// TwinCAT 3 PLC project PLC
// ProgramVersion: 3.1.4024.0
// libraries:
//   SPT Base Types, * (Beckhoff Automation LLC)
//   Tc2_Standard, * (Beckhoff Automation GmbH)
//   Tc2_System, * (Beckhoff Automation GmbH)
//   Tc3_Module, * (Beckhoff Automation GmbH)
//   Tc3_PackML_V2, * (Beckhoff Automation GmbH)
// project tree:
//   DUTs/HMI/ ST_HMI_Machine.TcDUT (not stored), ST_HMI_Machine_Command.TcDUT (not stored), ST_HMI_Machine_Config.TcDUT (not stored), ST_HMI_Machine_Status.TcDUT (not stored)
//   / GlobalTextList.TcGTLO, PlcTask.TcTTO, Visualization Manager.TcVMO (not stored)
//   GVLs/ gHMI.TcGVL
//   POUs/ MAIN.TcPOU
//   Templates/EM/ FB_EM_Template.TcPOU
//   VISUs/VFMs/ VFM_Machine.TcVIS (not stored), VFM_MachineControl.TcVIS (not stored), VFM_Module.TcVIS (not stored), VFM_OperatingMode.TcVIS (not stored), VFM_PackML.TcVIS (not stored), VFM_PackML_Manual.TcVIS (not stored)
//   VISUs/ VIS_Main.TcVIS (not stored)
//   _Machine/00_Machine/ FB_UM_Machine.TcPOU
//   _Machine/01_EM_Infeed/ FB_EM_Infeed.TcPOU
//   _Machine/02_EM_Work/ FB_EM_Work.TcPOU
//   _Machine/03_EM_Outfeed/ FB_EM_Outfeed.TcPOU
// real-time tasks:
//   TASK PlcTask: cycle T#10ms, priority 20, ADS port 350

CONFIGURATION PLC
    RESOURCE PLC ON TwinCAT3
        TASK PlcTask(INTERVAL := T#10ms, PRIORITY := 20);
        PROGRAM MAIN WITH PlcTask : MAIN;
    END_RESOURCE
END_CONFIGURATION

// ---- GVLs/gHMI.TcGVL
{attribute 'qualified_only'}
VAR_GLOBAL
END_VAR

// ---- POUs/MAIN.TcPOU
PROGRAM MAIN
VAR
	Machine: FB_UM_Machine	:= (Name := 'Machine', LogStateChanges := TRUE);
	Initialized: BOOL;
END_VAR

CyclicLogic();

METHOD CyclicLogic : BOOL
VAR_INPUT
END_VAR
IF NOT Initialized THEN
    Initialized := Initialize();
    RETURN;
END_IF

Machine.CyclicLogic();
END_METHOD

METHOD Initialize : BOOL
VAR_INPUT
END_VAR
Initialize := TRUE;
END_METHOD

END_PROGRAM

// ---- _Machine/00_Machine/FB_UM_Machine.TcPOU
FUNCTION_BLOCK FB_UM_Machine EXTENDS FB_PackML_BaseModule
VAR
	// Submodules
	EM_Infeed: 	FB_EM_Infeed 	:= (Name := 'Infeed', LogStateChanges := TRUE);
	EM_Work:	FB_EM_Work 		:= (Name := 'Work', LogStateChanges := TRUE);
	EM_Outfeed:	FB_EM_Outfeed 	:= (Name := 'Outfeed', LogStateChanges := TRUE);
	// Components
	
	// Module Data
	// --Param
	// --Recipe
	// --HMI
	HMI: ST_HMI_Machine;
	
	// Alarms
	
	// Other I/O

	// Machine Control
	rtrigControl: R_TRIG;
	CheckAbort: BOOL;
	CheckStop: BOOL;
	
	// Miscellaneous
	
END_VAR

METHOD PROTECTED Aborted
VAR_INPUT
END_VAR
END_METHOD

METHOD PROTECTED Aborting
VAR_INPUT
END_VAR
CASE _CurrentMode OF
	E_PMLUnitMode.ePMLUnitMode_Production:
        CASE DescendantSequenceState OF
			0:
				NoStateTasksToComplete := FALSE;
				DescendantSequenceState := DescendantSequenceState + 10;
			10:
				StateTasksComplete := TRUE;
		END_CASE
		
	E_PMLUnitMode.ePMLUnitMode_Manual, E_PMLUnitMode.ePMLUnitMode_Maintenance:
        ;	
END_CASE

// Call Super
SUPER^.Aborting();
END_METHOD

METHOD PROTECTED Clearing
VAR_INPUT
END_VAR
CASE _CurrentMode OF
	E_PMLUnitMode.ePMLUnitMode_Production:
        CASE DescendantSequenceState OF
			0:
				NoStateTasksToComplete := FALSE;
				DescendantSequenceState := DescendantSequenceState + 10;
			10:
				StateTasksComplete := TRUE;
		END_CASE
		
	E_PMLUnitMode.ePMLUnitMode_Manual, E_PMLUnitMode.ePMLUnitMode_Maintenance:
        ;	
END_CASE

// Call Super
SUPER^.Clearing();
END_METHOD

METHOD PROTECTED Complete
VAR_INPUT
END_VAR
END_METHOD

//! @summary Initializes event function blocks using this module's name
METHOD PROTECTED CreateEvents

//! @description This method is called by <c>Initialize()</c> as required
// Add your event creation here

// Super call to base
SUPER^.CreateEvents();
END_METHOD

METHOD CyclicLogic
VAR_INPUT
END_VAR
IF NOT _InitComplete THEN
    _InitComplete := Initialize();
    RETURN;
END_IF

MachineControl();

SUPER^.CyclicLogic();
END_METHOD

METHOD PROTECTED Execute
VAR_INPUT
END_VAR
CASE _CurrentMode OF
	E_PMLUnitMode.ePMLUnitMode_Production:
        CASE DescendantSequenceState OF
			0:
				DescendantSequenceState := DescendantSequenceState + 10;
			10:
				;
		END_CASE
		
	E_PMLUnitMode.ePMLUnitMode_Manual, E_PMLUnitMode.ePMLUnitMode_Maintenance:
        ;	
END_CASE
END_METHOD

METHOD PROTECTED Held
VAR_INPUT
END_VAR
END_METHOD

METHOD PROTECTED Holding
VAR_INPUT
END_VAR
CASE _CurrentMode OF
	E_PMLUnitMode.ePMLUnitMode_Production:
        CASE DescendantSequenceState OF
			0:
				NoStateTasksToComplete := FALSE;
				DescendantSequenceState := DescendantSequenceState + 10;
			10:
				StateTasksComplete := TRUE;
		END_CASE
		
	E_PMLUnitMode.ePMLUnitMode_Manual, E_PMLUnitMode.ePMLUnitMode_Maintenance:
        ;	
END_CASE

// Call Super
SUPER^.Holding();
END_METHOD

METHOD PROTECTED Idle
VAR_INPUT
END_VAR
END_METHOD

//! @summary Basic module initialization logic
METHOD PROTECTED Initialize : BOOL;
VAR
	i						 : UDINT;
	varInfo					 : __SYSTEM.VAR_INFO;
	AllSubUnitsInitialized	 : BOOL := TRUE;
	AllComponentsInitialized : BOOL := TRUE;
END_VAR

//! @description This method is called by <c>CyclicLogic()</c> as required
Initialize := FALSE;
CASE DescendantSequenceState OF
    0: // Initialize
        _LogModeChanges         := FALSE;
        _LogStateChanges        := FALSE;
        DescendantSequenceState := DescendantSequenceState + 10;
	
	10: // Register Submodules
		RegisterSubmodule(EM_Infeed);
		RegisterSubmodule(EM_Work);
		RegisterSubmodule(EM_Outfeed);
		DescendantSequenceState := DescendantSequenceState + 10;
		
    20: // Register Components
		//RegisterComponent(component);
        DescendantSequenceState := DescendantSequenceState + 10;
		
    30: // Call the Super
        IF SUPER^.Initialize() THEN
            DescendantSequenceState := DescendantSequenceState + 10;
        END_IF
    40:
        Initialize := TRUE;
END_CASE
END_METHOD

METHOD MachineControl
VAR_INPUT
END_VAR
// Control Triggers
rtrigControl(CLK:= HMI.Command.Start XOR HMI.Command.Stop XOR HMI.Command.Reset XOR HMI.Command.Abort);

CASE CurrentState OF
	E_PMLState.ePMLState_Aborting:
		CheckAbort := FALSE;
		CheckStop := FALSE;
		
	E_PMLState.ePMLState_Aborted:
		// Wait for Reset to Clear
		IF rtrigControl.Q AND HMI.Command.Reset THEN
			ChangeState(E_PMLCommand.ePMLCommand_Clear);
		END_IF
		
	E_PMLState.ePMLState_Clearing:
		CheckAbort := TRUE;
		CheckStop := FALSE;
		
	E_PMLState.ePMLState_Stopping:
		CheckAbort := TRUE;
		CheckStop := FALSE;
		
	E_PMLState.ePMLState_Stopped:
		// Wait for Reset
		IF rtrigControl.Q AND HMI.Command.Reset THEN
			ChangeState(E_PMLCommand.ePMLCommand_Reset);
		END_IF
		
	E_PMLState.ePMLState_Resetting:
		CheckAbort := TRUE;
		CheckStop := TRUE;
	
	E_PMLState.ePMLState_Idle:
		// Wait for Start
		IF rtrigControl.Q AND HMI.Command.Start THEN
			ChangeState(E_PMLCommand.ePMLCommand_Start);
		END_IF
	
END_CASE

// Check for Abort or Stop
IF rtrigControl.Q AND HMI.Command.Abort THEN
	ChangeState(E_PMLCommand.ePMLCommand_Abort);
ELSIF rtrigControl.Q AND HMI.Command.Stop THEN
	ChangeState(E_PMLCommand.ePMLCommand_Stop);
END_IF
END_METHOD

METHOD PROTECTED Resetting
VAR_INPUT
END_VAR
CASE _CurrentMode OF
	E_PMLUnitMode.ePMLUnitMode_Production:
        CASE DescendantSequenceState OF
			0:
				NoStateTasksToComplete := FALSE;
				DescendantSequenceState := DescendantSequenceState + 10;
			10:
				StateTasksComplete := TRUE;
		END_CASE
		
	E_PMLUnitMode.ePMLUnitMode_Manual, E_PMLUnitMode.ePMLUnitMode_Maintenance:
        ;	
END_CASE

// Call Super
SUPER^.Resetting();
END_METHOD

METHOD PROTECTED Starting
VAR_INPUT
END_VAR
CASE _CurrentMode OF
	E_PMLUnitMode.ePMLUnitMode_Production:
        CASE DescendantSequenceState OF
			0:
				NoStateTasksToComplete := FALSE;
				DescendantSequenceState := DescendantSequenceState + 10;
			10:
				StateTasksComplete := TRUE;
		END_CASE
		
	E_PMLUnitMode.ePMLUnitMode_Manual, E_PMLUnitMode.ePMLUnitMode_Maintenance:
        ;	
END_CASE

// Call Super
SUPER^.Starting();
END_METHOD

METHOD PROTECTED Stopped
VAR_INPUT
END_VAR
END_METHOD

METHOD PROTECTED Stopping
VAR_INPUT
END_VAR
CASE _CurrentMode OF
	E_PMLUnitMode.ePMLUnitMode_Production:
        CASE DescendantSequenceState OF
			0:
				NoStateTasksToComplete := FALSE;
				DescendantSequenceState := DescendantSequenceState + 10;
			10:
				StateTasksComplete := TRUE;
		END_CASE
		
	E_PMLUnitMode.ePMLUnitMode_Manual, E_PMLUnitMode.ePMLUnitMode_Maintenance:
        ;	
END_CASE

// Call Super
SUPER^.Stopping();
END_METHOD

METHOD PROTECTED Suspended
VAR_INPUT
END_VAR
END_METHOD

METHOD PROTECTED Suspending
VAR_INPUT
END_VAR
CASE _CurrentMode OF
	E_PMLUnitMode.ePMLUnitMode_Production:
        CASE DescendantSequenceState OF
			0:
				NoStateTasksToComplete := FALSE;
				DescendantSequenceState := DescendantSequenceState + 10;
			10:
				StateTasksComplete := TRUE;
		END_CASE
		
	E_PMLUnitMode.ePMLUnitMode_Manual, E_PMLUnitMode.ePMLUnitMode_Maintenance:
        ;	
END_CASE

// Call Super
SUPER^.Suspending();
END_METHOD

METHOD PROTECTED Undefined
VAR_INPUT
END_VAR
END_METHOD

METHOD PROTECTED Unholding
VAR_INPUT
END_VAR
CASE _CurrentMode OF
	E_PMLUnitMode.ePMLUnitMode_Production:
        CASE DescendantSequenceState OF
			0:
				NoStateTasksToComplete := FALSE;
				DescendantSequenceState := DescendantSequenceState + 10;
			10:
				StateTasksComplete := TRUE;
		END_CASE
		
	E_PMLUnitMode.ePMLUnitMode_Manual, E_PMLUnitMode.ePMLUnitMode_Maintenance:
        ;	
END_CASE

// Call Super
SUPER^.Unholding();
END_METHOD

METHOD PROTECTED Unsuspending
VAR_INPUT
END_VAR
CASE _CurrentMode OF
	E_PMLUnitMode.ePMLUnitMode_Production:
        CASE DescendantSequenceState OF
			0:
				NoStateTasksToComplete := FALSE;
				DescendantSequenceState := DescendantSequenceState + 10;
			10:
				StateTasksComplete := TRUE;
		END_CASE
		
	E_PMLUnitMode.ePMLUnitMode_Manual, E_PMLUnitMode.ePMLUnitMode_Maintenance:
        ;	
END_CASE

// Call Super
SUPER^.Unsuspending();
END_METHOD

END_FUNCTION_BLOCK

// ---- _Machine/01_EM_Infeed/FB_EM_Infeed.TcPOU
FUNCTION_BLOCK FB_EM_Infeed EXTENDS FB_PackML_BaseModule
VAR
	// Submodules
	
	// Components
	
	// Module Data
	// --Param
	// --Recipe
	// --HMI
	
	// Alarms
	
	// Other I/O
	
	// Miscellaneous
	
END_VAR

METHOD PROTECTED Aborted
VAR_INPUT
END_VAR
END_METHOD

METHOD PROTECTED Aborting
VAR_INPUT
END_VAR
CASE _CurrentMode OF
	E_PMLUnitMode.ePMLUnitMode_Production:
        CASE DescendantSequenceState OF
			0:
				NoStateTasksToComplete := FALSE;
				DescendantSequenceState := DescendantSequenceState + 10;
			10:
				StateTasksComplete := TRUE;
		END_CASE
		
	E_PMLUnitMode.ePMLUnitMode_Manual, E_PMLUnitMode.ePMLUnitMode_Maintenance:
        ;	
END_CASE

// Call Super
SUPER^.Aborting();
END_METHOD

METHOD PROTECTED Clearing
VAR_INPUT
END_VAR
CASE _CurrentMode OF
	E_PMLUnitMode.ePMLUnitMode_Production:
        CASE DescendantSequenceState OF
			0:
				NoStateTasksToComplete := FALSE;
				DescendantSequenceState := DescendantSequenceState + 10;
			10:
				StateTasksComplete := TRUE;
		END_CASE
		
	E_PMLUnitMode.ePMLUnitMode_Manual, E_PMLUnitMode.ePMLUnitMode_Maintenance:
        ;	
END_CASE

// Call Super
SUPER^.Clearing();
END_METHOD

METHOD PROTECTED Complete
VAR_INPUT
END_VAR
END_METHOD

//! @summary Initializes event function blocks using this module's name
METHOD PROTECTED CreateEvents

//! @description This method is called by <c>Initialize()</c> as required
// Add your event creation here

// Super call to base
SUPER^.CreateEvents();
END_METHOD

METHOD CyclicLogic
VAR_INPUT
END_VAR
IF NOT _InitComplete THEN
    _InitComplete := Initialize();
    RETURN;
END_IF

SUPER^.CyclicLogic();
END_METHOD

METHOD PROTECTED Execute
VAR_INPUT
END_VAR
CASE _CurrentMode OF
	E_PMLUnitMode.ePMLUnitMode_Production:
        CASE DescendantSequenceState OF
			0:
				DescendantSequenceState := DescendantSequenceState + 10;
			10:
				;
		END_CASE
		
	E_PMLUnitMode.ePMLUnitMode_Manual, E_PMLUnitMode.ePMLUnitMode_Maintenance:
        ;	
END_CASE
END_METHOD

METHOD PROTECTED Held
VAR_INPUT
END_VAR
END_METHOD

METHOD PROTECTED Holding
VAR_INPUT
END_VAR
CASE _CurrentMode OF
	E_PMLUnitMode.ePMLUnitMode_Production:
        CASE DescendantSequenceState OF
			0:
				NoStateTasksToComplete := FALSE;
				DescendantSequenceState := DescendantSequenceState + 10;
			10:
				StateTasksComplete := TRUE;
		END_CASE
		
	E_PMLUnitMode.ePMLUnitMode_Manual, E_PMLUnitMode.ePMLUnitMode_Maintenance:
        ;	
END_CASE

// Call Super
SUPER^.Holding();
END_METHOD

METHOD PROTECTED Idle
VAR_INPUT
END_VAR
END_METHOD

//! @summary Basic module initialization logic
METHOD PROTECTED Initialize : BOOL;
VAR
	i						 : UDINT;
	varInfo					 : __SYSTEM.VAR_INFO;
	AllSubUnitsInitialized	 : BOOL := TRUE;
	AllComponentsInitialized : BOOL := TRUE;
END_VAR

//! @description This method is called by <c>CyclicLogic()</c> as required
Initialize := FALSE;
CASE DescendantSequenceState OF
    0: // Initialize
        _LogModeChanges         := FALSE;
        _LogStateChanges        := FALSE;
        DescendantSequenceState := DescendantSequenceState + 10;
	
	10: // Register Submodules
		//RegisterSubmodule(submodule);
		DescendantSequenceState := DescendantSequenceState + 10;
    20: // Register Components
		//RegisterComponent(component);
        DescendantSequenceState := DescendantSequenceState + 10;
    30: // Call the Super
        IF SUPER^.Initialize() THEN
            DescendantSequenceState := DescendantSequenceState + 10;
        END_IF
    40:
        Initialize := TRUE;
END_CASE
END_METHOD

METHOD PROTECTED Resetting
VAR_INPUT
END_VAR
CASE _CurrentMode OF
	E_PMLUnitMode.ePMLUnitMode_Production:
        CASE DescendantSequenceState OF
			0:
				NoStateTasksToComplete := FALSE;
				DescendantSequenceState := DescendantSequenceState + 10;
			10:
				StateTasksComplete := TRUE;
		END_CASE
		
	E_PMLUnitMode.ePMLUnitMode_Manual, E_PMLUnitMode.ePMLUnitMode_Maintenance:
        ;	
END_CASE

// Call Super
SUPER^.Resetting();
END_METHOD

METHOD PROTECTED Starting
VAR_INPUT
END_VAR
CASE _CurrentMode OF
	E_PMLUnitMode.ePMLUnitMode_Production:
        CASE DescendantSequenceState OF
			0:
				NoStateTasksToComplete := FALSE;
				DescendantSequenceState := DescendantSequenceState + 10;
			10:
				StateTasksComplete := TRUE;
		END_CASE
		
	E_PMLUnitMode.ePMLUnitMode_Manual, E_PMLUnitMode.ePMLUnitMode_Maintenance:
        ;	
END_CASE

// Call Super
SUPER^.Starting();
END_METHOD

METHOD PROTECTED Stopped
VAR_INPUT
END_VAR
END_METHOD

METHOD PROTECTED Stopping
VAR_INPUT
END_VAR
CASE _CurrentMode OF
	E_PMLUnitMode.ePMLUnitMode_Production:
        CASE DescendantSequenceState OF
			0:
				NoStateTasksToComplete := FALSE;
				DescendantSequenceState := DescendantSequenceState + 10;
			10:
				StateTasksComplete := TRUE;
		END_CASE
		
	E_PMLUnitMode.ePMLUnitMode_Manual, E_PMLUnitMode.ePMLUnitMode_Maintenance:
        ;	
END_CASE

// Call Super
SUPER^.Stopping();
END_METHOD

METHOD PROTECTED Suspended
VAR_INPUT
END_VAR
END_METHOD

METHOD PROTECTED Suspending
VAR_INPUT
END_VAR
CASE _CurrentMode OF
	E_PMLUnitMode.ePMLUnitMode_Production:
        CASE DescendantSequenceState OF
			0:
				NoStateTasksToComplete := FALSE;
				DescendantSequenceState := DescendantSequenceState + 10;
			10:
				StateTasksComplete := TRUE;
		END_CASE
		
	E_PMLUnitMode.ePMLUnitMode_Manual, E_PMLUnitMode.ePMLUnitMode_Maintenance:
        ;	
END_CASE

// Call Super
SUPER^.Suspending();
END_METHOD

METHOD PROTECTED Undefined
VAR_INPUT
END_VAR
END_METHOD

METHOD PROTECTED Unholding
VAR_INPUT
END_VAR
CASE _CurrentMode OF
	E_PMLUnitMode.ePMLUnitMode_Production:
        CASE DescendantSequenceState OF
			0:
				NoStateTasksToComplete := FALSE;
				DescendantSequenceState := DescendantSequenceState + 10;
			10:
				StateTasksComplete := TRUE;
		END_CASE
		
	E_PMLUnitMode.ePMLUnitMode_Manual, E_PMLUnitMode.ePMLUnitMode_Maintenance:
        ;	
END_CASE

// Call Super
SUPER^.Unholding();
END_METHOD

METHOD PROTECTED Unsuspending
VAR_INPUT
END_VAR
CASE _CurrentMode OF
	E_PMLUnitMode.ePMLUnitMode_Production:
        CASE DescendantSequenceState OF
			0:
				NoStateTasksToComplete := FALSE;
				DescendantSequenceState := DescendantSequenceState + 10;
			10:
				StateTasksComplete := TRUE;
		END_CASE
		
	E_PMLUnitMode.ePMLUnitMode_Manual, E_PMLUnitMode.ePMLUnitMode_Maintenance:
        ;	
END_CASE

// Call Super
SUPER^.Unsuspending();
END_METHOD

END_FUNCTION_BLOCK

// ---- _Machine/02_EM_Work/FB_EM_Work.TcPOU
FUNCTION_BLOCK FB_EM_Work EXTENDS FB_PackML_BaseModule
VAR
	// Submodules
	
	// Components
	
	// Module Data
	// --Param
	// --Recipe
	// --HMI
	
	// Alarms
	
	// Other I/O
	
	// Miscellaneous
	
END_VAR

METHOD PROTECTED Aborted
VAR_INPUT
END_VAR
END_METHOD

METHOD PROTECTED Aborting
VAR_INPUT
END_VAR
CASE _CurrentMode OF
	E_PMLUnitMode.ePMLUnitMode_Production:
        CASE DescendantSequenceState OF
			0:
				NoStateTasksToComplete := FALSE;
				DescendantSequenceState := DescendantSequenceState + 10;
			10:
				StateTasksComplete := TRUE;
		END_CASE
		
	E_PMLUnitMode.ePMLUnitMode_Manual, E_PMLUnitMode.ePMLUnitMode_Maintenance:
        ;	
END_CASE

// Call Super
SUPER^.Aborting();
END_METHOD

METHOD PROTECTED Clearing
VAR_INPUT
END_VAR
CASE _CurrentMode OF
	E_PMLUnitMode.ePMLUnitMode_Production:
        CASE DescendantSequenceState OF
			0:
				NoStateTasksToComplete := FALSE;
				DescendantSequenceState := DescendantSequenceState + 10;
			10:
				StateTasksComplete := TRUE;
		END_CASE
		
	E_PMLUnitMode.ePMLUnitMode_Manual, E_PMLUnitMode.ePMLUnitMode_Maintenance:
        ;	
END_CASE

// Call Super
SUPER^.Clearing();
END_METHOD

METHOD PROTECTED Complete
VAR_INPUT
END_VAR
END_METHOD

//! @summary Initializes event function blocks using this module's name
METHOD PROTECTED CreateEvents

//! @description This method is called by <c>Initialize()</c> as required
// Add your event creation here

// Super call to base
SUPER^.CreateEvents();
END_METHOD

METHOD CyclicLogic
VAR_INPUT
END_VAR
IF NOT _InitComplete THEN
    _InitComplete := Initialize();
    RETURN;
END_IF

SUPER^.CyclicLogic();
END_METHOD

METHOD PROTECTED Execute
VAR_INPUT
END_VAR
CASE _CurrentMode OF
	E_PMLUnitMode.ePMLUnitMode_Production:
        CASE DescendantSequenceState OF
			0:
				DescendantSequenceState := DescendantSequenceState + 10;
			10:
				;
		END_CASE
		
	E_PMLUnitMode.ePMLUnitMode_Manual, E_PMLUnitMode.ePMLUnitMode_Maintenance:
        ;	
END_CASE
END_METHOD

METHOD PROTECTED Held
VAR_INPUT
END_VAR
END_METHOD

METHOD PROTECTED Holding
VAR_INPUT
END_VAR
CASE _CurrentMode OF
	E_PMLUnitMode.ePMLUnitMode_Production:
        CASE DescendantSequenceState OF
			0:
				NoStateTasksToComplete := FALSE;
				DescendantSequenceState := DescendantSequenceState + 10;
			10:
				StateTasksComplete := TRUE;
		END_CASE
		
	E_PMLUnitMode.ePMLUnitMode_Manual, E_PMLUnitMode.ePMLUnitMode_Maintenance:
        ;	
END_CASE

// Call Super
SUPER^.Holding();
END_METHOD

METHOD PROTECTED Idle
VAR_INPUT
END_VAR
END_METHOD

//! @summary Basic module initialization logic
METHOD PROTECTED Initialize : BOOL;
VAR
	i						 : UDINT;
	varInfo					 : __SYSTEM.VAR_INFO;
	AllSubUnitsInitialized	 : BOOL := TRUE;
	AllComponentsInitialized : BOOL := TRUE;
END_VAR

//! @description This method is called by <c>CyclicLogic()</c> as required
Initialize := FALSE;
CASE DescendantSequenceState OF
    0: // Initialize
        _LogModeChanges         := FALSE;
        _LogStateChanges        := FALSE;
        DescendantSequenceState := DescendantSequenceState + 10;
	
	10: // Register Submodules
		//RegisterSubmodule(submodule);
		DescendantSequenceState := DescendantSequenceState + 10;
    20: // Register Components
		//RegisterComponent(component);
        DescendantSequenceState := DescendantSequenceState + 10;
    30: // Call the Super
        IF SUPER^.Initialize() THEN
            DescendantSequenceState := DescendantSequenceState + 10;
        END_IF
    40:
        Initialize := TRUE;
END_CASE
END_METHOD

METHOD PROTECTED Resetting
VAR_INPUT
END_VAR
CASE _CurrentMode OF
	E_PMLUnitMode.ePMLUnitMode_Production:
        CASE DescendantSequenceState OF
			0:
				NoStateTasksToComplete := FALSE;
				DescendantSequenceState := DescendantSequenceState + 10;
			10:
				StateTasksComplete := TRUE;
		END_CASE
		
	E_PMLUnitMode.ePMLUnitMode_Manual, E_PMLUnitMode.ePMLUnitMode_Maintenance:
        ;	
END_CASE

// Call Super
SUPER^.Resetting();
END_METHOD

METHOD PROTECTED Starting
VAR_INPUT
END_VAR
CASE _CurrentMode OF
	E_PMLUnitMode.ePMLUnitMode_Production:
        CASE DescendantSequenceState OF
			0:
				NoStateTasksToComplete := FALSE;
				DescendantSequenceState := DescendantSequenceState + 10;
			10:
				StateTasksComplete := TRUE;
		END_CASE
		
	E_PMLUnitMode.ePMLUnitMode_Manual, E_PMLUnitMode.ePMLUnitMode_Maintenance:
        ;	
END_CASE

// Call Super
SUPER^.Starting();
END_METHOD

METHOD PROTECTED Stopped
VAR_INPUT
END_VAR
END_METHOD

METHOD PROTECTED Stopping
VAR_INPUT
END_VAR
CASE _CurrentMode OF
	E_PMLUnitMode.ePMLUnitMode_Production:
        CASE DescendantSequenceState OF
			0:
				NoStateTasksToComplete := FALSE;
				DescendantSequenceState := DescendantSequenceState + 10;
			10:
				StateTasksComplete := TRUE;
		END_CASE
		
	E_PMLUnitMode.ePMLUnitMode_Manual, E_PMLUnitMode.ePMLUnitMode_Maintenance:
        ;	
END_CASE

// Call Super
SUPER^.Stopping();
END_METHOD

METHOD PROTECTED Suspended
VAR_INPUT
END_VAR
END_METHOD

METHOD PROTECTED Suspending
VAR_INPUT
END_VAR
CASE _CurrentMode OF
	E_PMLUnitMode.ePMLUnitMode_Production:
        CASE DescendantSequenceState OF
			0:
				NoStateTasksToComplete := FALSE;
				DescendantSequenceState := DescendantSequenceState + 10;
			10:
				StateTasksComplete := TRUE;
		END_CASE
		
	E_PMLUnitMode.ePMLUnitMode_Manual, E_PMLUnitMode.ePMLUnitMode_Maintenance:
        ;	
END_CASE

// Call Super
SUPER^.Suspending();
END_METHOD

METHOD PROTECTED Undefined
VAR_INPUT
END_VAR
END_METHOD

METHOD PROTECTED Unholding
VAR_INPUT
END_VAR
CASE _CurrentMode OF
	E_PMLUnitMode.ePMLUnitMode_Production:
        CASE DescendantSequenceState OF
			0:
				NoStateTasksToComplete := FALSE;
				DescendantSequenceState := DescendantSequenceState + 10;
			10:
				StateTasksComplete := TRUE;
		END_CASE
		
	E_PMLUnitMode.ePMLUnitMode_Manual, E_PMLUnitMode.ePMLUnitMode_Maintenance:
        ;	
END_CASE

// Call Super
SUPER^.Unholding();
END_METHOD

METHOD PROTECTED Unsuspending
VAR_INPUT
END_VAR
CASE _CurrentMode OF
	E_PMLUnitMode.ePMLUnitMode_Production:
        CASE DescendantSequenceState OF
			0:
				NoStateTasksToComplete := FALSE;
				DescendantSequenceState := DescendantSequenceState + 10;
			10:
				StateTasksComplete := TRUE;
		END_CASE
		
	E_PMLUnitMode.ePMLUnitMode_Manual, E_PMLUnitMode.ePMLUnitMode_Maintenance:
        ;	
END_CASE

// Call Super
SUPER^.Unsuspending();
END_METHOD

END_FUNCTION_BLOCK

// ---- _Machine/03_EM_Outfeed/FB_EM_Outfeed.TcPOU
FUNCTION_BLOCK FB_EM_Outfeed EXTENDS FB_PackML_BaseModule
VAR
	// Submodules
	
	// Components
	
	// Module Data
	// --Param
	// --Recipe
	// --HMI
	
	// Alarms
	
	// Other I/O
	
	// Miscellaneous
	
END_VAR

METHOD PROTECTED Aborted
VAR_INPUT
END_VAR
END_METHOD

METHOD PROTECTED Aborting
VAR_INPUT
END_VAR
CASE _CurrentMode OF
	E_PMLUnitMode.ePMLUnitMode_Production:
        CASE DescendantSequenceState OF
			0:
				NoStateTasksToComplete := FALSE;
				DescendantSequenceState := DescendantSequenceState + 10;
			10:
				StateTasksComplete := TRUE;
		END_CASE
		
	E_PMLUnitMode.ePMLUnitMode_Manual, E_PMLUnitMode.ePMLUnitMode_Maintenance:
        ;	
END_CASE

// Call Super
SUPER^.Aborting();
END_METHOD

METHOD PROTECTED Clearing
VAR_INPUT
END_VAR
CASE _CurrentMode OF
	E_PMLUnitMode.ePMLUnitMode_Production:
        CASE DescendantSequenceState OF
			0:
				NoStateTasksToComplete := FALSE;
				DescendantSequenceState := DescendantSequenceState + 10;
			10:
				StateTasksComplete := TRUE;
		END_CASE
		
	E_PMLUnitMode.ePMLUnitMode_Manual, E_PMLUnitMode.ePMLUnitMode_Maintenance:
        ;	
END_CASE

// Call Super
SUPER^.Clearing();
END_METHOD

METHOD PROTECTED Complete
VAR_INPUT
END_VAR
END_METHOD

//! @summary Initializes event function blocks using this module's name
METHOD PROTECTED CreateEvents

//! @description This method is called by <c>Initialize()</c> as required
// Add your event creation here

// Super call to base
SUPER^.CreateEvents();
END_METHOD

METHOD CyclicLogic
VAR_INPUT
END_VAR
IF NOT _InitComplete THEN
    _InitComplete := Initialize();
    RETURN;
END_IF

SUPER^.CyclicLogic();
END_METHOD

METHOD PROTECTED Execute
VAR_INPUT
END_VAR
CASE _CurrentMode OF
	E_PMLUnitMode.ePMLUnitMode_Production:
        CASE DescendantSequenceState OF
			0:
				DescendantSequenceState := DescendantSequenceState + 10;
			10:
				;
		END_CASE
		
	E_PMLUnitMode.ePMLUnitMode_Manual, E_PMLUnitMode.ePMLUnitMode_Maintenance:
        ;	
END_CASE
END_METHOD

METHOD PROTECTED Held
VAR_INPUT
END_VAR
END_METHOD

METHOD PROTECTED Holding
VAR_INPUT
END_VAR
CASE _CurrentMode OF
	E_PMLUnitMode.ePMLUnitMode_Production:
        CASE DescendantSequenceState OF
			0:
				NoStateTasksToComplete := FALSE;
				DescendantSequenceState := DescendantSequenceState + 10;
			10:
				StateTasksComplete := TRUE;
		END_CASE
		
	E_PMLUnitMode.ePMLUnitMode_Manual, E_PMLUnitMode.ePMLUnitMode_Maintenance:
        ;	
END_CASE

// Call Super
SUPER^.Holding();
END_METHOD

METHOD PROTECTED Idle
VAR_INPUT
END_VAR
END_METHOD

//! @summary Basic module initialization logic
METHOD PROTECTED Initialize : BOOL;
VAR
	i						 : UDINT;
	varInfo					 : __SYSTEM.VAR_INFO;
	AllSubUnitsInitialized	 : BOOL := TRUE;
	AllComponentsInitialized : BOOL := TRUE;
END_VAR

//! @description This method is called by <c>CyclicLogic()</c> as required
Initialize := FALSE;
CASE DescendantSequenceState OF
    0: // Initialize
        _LogModeChanges         := FALSE;
        _LogStateChanges        := FALSE;
        DescendantSequenceState := DescendantSequenceState + 10;
	
	10: // Register Submodules
		//RegisterSubmodule(submodule);
		DescendantSequenceState := DescendantSequenceState + 10;
    20: // Register Components
		//RegisterComponent(component);
        DescendantSequenceState := DescendantSequenceState + 10;
    30: // Call the Super
        IF SUPER^.Initialize() THEN
            DescendantSequenceState := DescendantSequenceState + 10;
        END_IF
    40:
        Initialize := TRUE;
END_CASE
END_METHOD

METHOD PROTECTED Resetting
VAR_INPUT
END_VAR
CASE _CurrentMode OF
	E_PMLUnitMode.ePMLUnitMode_Production:
        CASE DescendantSequenceState OF
			0:
				NoStateTasksToComplete := FALSE;
				DescendantSequenceState := DescendantSequenceState + 10;
			10:
				StateTasksComplete := TRUE;
		END_CASE
		
	E_PMLUnitMode.ePMLUnitMode_Manual, E_PMLUnitMode.ePMLUnitMode_Maintenance:
        ;	
END_CASE

// Call Super
SUPER^.Resetting();
END_METHOD

METHOD PROTECTED Starting
VAR_INPUT
END_VAR
CASE _CurrentMode OF
	E_PMLUnitMode.ePMLUnitMode_Production:
        CASE DescendantSequenceState OF
			0:
				NoStateTasksToComplete := FALSE;
				DescendantSequenceState := DescendantSequenceState + 10;
			10:
				StateTasksComplete := TRUE;
		END_CASE
		
	E_PMLUnitMode.ePMLUnitMode_Manual, E_PMLUnitMode.ePMLUnitMode_Maintenance:
        ;	
END_CASE

// Call Super
SUPER^.Starting();
END_METHOD

METHOD PROTECTED Stopped
VAR_INPUT
END_VAR
END_METHOD

METHOD PROTECTED Stopping
VAR_INPUT
END_VAR
CASE _CurrentMode OF
	E_PMLUnitMode.ePMLUnitMode_Production:
        CASE DescendantSequenceState OF
			0:
				NoStateTasksToComplete := FALSE;
				DescendantSequenceState := DescendantSequenceState + 10;
			10:
				StateTasksComplete := TRUE;
		END_CASE
		
	E_PMLUnitMode.ePMLUnitMode_Manual, E_PMLUnitMode.ePMLUnitMode_Maintenance:
        ;	
END_CASE

// Call Super
SUPER^.Stopping();
END_METHOD

METHOD PROTECTED Suspended
VAR_INPUT
END_VAR
END_METHOD

METHOD PROTECTED Suspending
VAR_INPUT
END_VAR
CASE _CurrentMode OF
	E_PMLUnitMode.ePMLUnitMode_Production:
        CASE DescendantSequenceState OF
			0:
				NoStateTasksToComplete := FALSE;
				DescendantSequenceState := DescendantSequenceState + 10;
			10:
				StateTasksComplete := TRUE;
		END_CASE
		
	E_PMLUnitMode.ePMLUnitMode_Manual, E_PMLUnitMode.ePMLUnitMode_Maintenance:
        ;	
END_CASE

// Call Super
SUPER^.Suspending();
END_METHOD

METHOD PROTECTED Undefined
VAR_INPUT
END_VAR
END_METHOD

METHOD PROTECTED Unholding
VAR_INPUT
END_VAR
CASE _CurrentMode OF
	E_PMLUnitMode.ePMLUnitMode_Production:
        CASE DescendantSequenceState OF
			0:
				NoStateTasksToComplete := FALSE;
				DescendantSequenceState := DescendantSequenceState + 10;
			10:
				StateTasksComplete := TRUE;
		END_CASE
		
	E_PMLUnitMode.ePMLUnitMode_Manual, E_PMLUnitMode.ePMLUnitMode_Maintenance:
        ;	
END_CASE

// Call Super
SUPER^.Unholding();
END_METHOD

METHOD PROTECTED Unsuspending
VAR_INPUT
END_VAR
CASE _CurrentMode OF
	E_PMLUnitMode.ePMLUnitMode_Production:
        CASE DescendantSequenceState OF
			0:
				NoStateTasksToComplete := FALSE;
				DescendantSequenceState := DescendantSequenceState + 10;
			10:
				StateTasksComplete := TRUE;
		END_CASE
		
	E_PMLUnitMode.ePMLUnitMode_Manual, E_PMLUnitMode.ePMLUnitMode_Maintenance:
        ;	
END_CASE

// Call Super
SUPER^.Unsuspending();
END_METHOD

END_FUNCTION_BLOCK

// ---- Templates/EM/FB_EM_Template.TcPOU
FUNCTION_BLOCK FB_EM_Template EXTENDS FB_PackML_BaseModule
VAR
	// Submodules
	
	// Components
	
	// Module Data
	// --Param
	// --Recipe
	// --HMI
	
	// Alarms
	
	// Other I/O
	
	// Miscellaneous
	
END_VAR

METHOD PROTECTED Aborted
VAR_INPUT
END_VAR
END_METHOD

METHOD PROTECTED Aborting
VAR_INPUT
END_VAR
CASE _CurrentMode OF
	E_PMLUnitMode.ePMLUnitMode_Production:
        CASE DescendantSequenceState OF
			0:
				NoStateTasksToComplete := FALSE;
				DescendantSequenceState := DescendantSequenceState + 10;
			10:
				StateTasksComplete := TRUE;
		END_CASE
		
	E_PMLUnitMode.ePMLUnitMode_Manual, E_PMLUnitMode.ePMLUnitMode_Maintenance:
        ;	
END_CASE

// Call Super
SUPER^.Aborting();
END_METHOD

METHOD PROTECTED Clearing
VAR_INPUT
END_VAR
CASE _CurrentMode OF
	E_PMLUnitMode.ePMLUnitMode_Production:
        CASE DescendantSequenceState OF
			0:
				NoStateTasksToComplete := FALSE;
				DescendantSequenceState := DescendantSequenceState + 10;
			10:
				StateTasksComplete := TRUE;
		END_CASE
		
	E_PMLUnitMode.ePMLUnitMode_Manual, E_PMLUnitMode.ePMLUnitMode_Maintenance:
        ;	
END_CASE

// Call Super
SUPER^.Clearing();
END_METHOD

METHOD PROTECTED Complete
VAR_INPUT
END_VAR
END_METHOD

//! @summary Initializes event function blocks using this module's name
METHOD PROTECTED CreateEvents

//! @description This method is called by <c>Initialize()</c> as required
// Add your event creation here

// Super call to base
SUPER^.CreateEvents();
END_METHOD

METHOD CyclicLogic
VAR_INPUT
END_VAR
IF NOT _InitComplete THEN
    _InitComplete := Initialize();
    RETURN;
END_IF

SUPER^.CyclicLogic();
END_METHOD

METHOD PROTECTED Execute
VAR_INPUT
END_VAR
CASE _CurrentMode OF
	E_PMLUnitMode.ePMLUnitMode_Production:
        CASE DescendantSequenceState OF
			0:
				DescendantSequenceState := DescendantSequenceState + 10;
			10:
				;
		END_CASE
		
	E_PMLUnitMode.ePMLUnitMode_Manual, E_PMLUnitMode.ePMLUnitMode_Maintenance:
        ;	
END_CASE
END_METHOD

METHOD PROTECTED Held
VAR_INPUT
END_VAR
END_METHOD

METHOD PROTECTED Holding
VAR_INPUT
END_VAR
CASE _CurrentMode OF
	E_PMLUnitMode.ePMLUnitMode_Production:
        CASE DescendantSequenceState OF
			0:
				NoStateTasksToComplete := FALSE;
				DescendantSequenceState := DescendantSequenceState + 10;
			10:
				StateTasksComplete := TRUE;
		END_CASE
		
	E_PMLUnitMode.ePMLUnitMode_Manual, E_PMLUnitMode.ePMLUnitMode_Maintenance:
        ;	
END_CASE

// Call Super
SUPER^.Holding();
END_METHOD

METHOD PROTECTED Idle
VAR_INPUT
END_VAR
END_METHOD

//! @summary Basic module initialization logic
METHOD PROTECTED Initialize : BOOL;
VAR
	i						 : UDINT;
	varInfo					 : __SYSTEM.VAR_INFO;
	AllSubUnitsInitialized	 : BOOL := TRUE;
	AllComponentsInitialized : BOOL := TRUE;
END_VAR

//! @description This method is called by <c>CyclicLogic()</c> as required
Initialize := FALSE;
CASE DescendantSequenceState OF
    0: // Initialize
        _LogModeChanges         := FALSE;
        _LogStateChanges        := FALSE;
        DescendantSequenceState := DescendantSequenceState + 10;
	
	10: // Register Submodules
		//RegisterSubmodule(submodule);
		DescendantSequenceState := DescendantSequenceState + 10;
    20: // Register Components
		//RegisterComponent(component);
        DescendantSequenceState := DescendantSequenceState + 10;
    30: // Call the Super
        IF SUPER^.Initialize() THEN
            DescendantSequenceState := DescendantSequenceState + 10;
        END_IF
    40:
        Initialize := TRUE;
END_CASE
END_METHOD

METHOD PROTECTED Resetting
VAR_INPUT
END_VAR
CASE _CurrentMode OF
	E_PMLUnitMode.ePMLUnitMode_Production:
        CASE DescendantSequenceState OF
			0:
				NoStateTasksToComplete := FALSE;
				DescendantSequenceState := DescendantSequenceState + 10;
			10:
				StateTasksComplete := TRUE;
		END_CASE
		
	E_PMLUnitMode.ePMLUnitMode_Manual, E_PMLUnitMode.ePMLUnitMode_Maintenance:
        ;	
END_CASE

// Call Super
SUPER^.Resetting();
END_METHOD

METHOD PROTECTED Starting
VAR_INPUT
END_VAR
CASE _CurrentMode OF
	E_PMLUnitMode.ePMLUnitMode_Production:
        CASE DescendantSequenceState OF
			0:
				NoStateTasksToComplete := FALSE;
				DescendantSequenceState := DescendantSequenceState + 10;
			10:
				StateTasksComplete := TRUE;
		END_CASE
		
	E_PMLUnitMode.ePMLUnitMode_Manual, E_PMLUnitMode.ePMLUnitMode_Maintenance:
        ;	
END_CASE

// Call Super
SUPER^.Starting();
END_METHOD

METHOD PROTECTED Stopped
VAR_INPUT
END_VAR
END_METHOD

METHOD PROTECTED Stopping
VAR_INPUT
END_VAR
CASE _CurrentMode OF
	E_PMLUnitMode.ePMLUnitMode_Production:
        CASE DescendantSequenceState OF
			0:
				NoStateTasksToComplete := FALSE;
				DescendantSequenceState := DescendantSequenceState + 10;
			10:
				StateTasksComplete := TRUE;
		END_CASE
		
	E_PMLUnitMode.ePMLUnitMode_Manual, E_PMLUnitMode.ePMLUnitMode_Maintenance:
        ;	
END_CASE

// Call Super
SUPER^.Stopping();
END_METHOD

METHOD PROTECTED Suspended
VAR_INPUT
END_VAR
END_METHOD

METHOD PROTECTED Suspending
VAR_INPUT
END_VAR
CASE _CurrentMode OF
	E_PMLUnitMode.ePMLUnitMode_Production:
        CASE DescendantSequenceState OF
			0:
				NoStateTasksToComplete := FALSE;
				DescendantSequenceState := DescendantSequenceState + 10;
			10:
				StateTasksComplete := TRUE;
		END_CASE
		
	E_PMLUnitMode.ePMLUnitMode_Manual, E_PMLUnitMode.ePMLUnitMode_Maintenance:
        ;	
END_CASE

// Call Super
SUPER^.Suspending();
END_METHOD

METHOD PROTECTED Undefined
VAR_INPUT
END_VAR
END_METHOD

METHOD PROTECTED Unholding
VAR_INPUT
END_VAR
CASE _CurrentMode OF
	E_PMLUnitMode.ePMLUnitMode_Production:
        CASE DescendantSequenceState OF
			0:
				NoStateTasksToComplete := FALSE;
				DescendantSequenceState := DescendantSequenceState + 10;
			10:
				StateTasksComplete := TRUE;
		END_CASE
		
	E_PMLUnitMode.ePMLUnitMode_Manual, E_PMLUnitMode.ePMLUnitMode_Maintenance:
        ;	
END_CASE

// Call Super
SUPER^.Unholding();
END_METHOD

METHOD PROTECTED Unsuspending
VAR_INPUT
END_VAR
CASE _CurrentMode OF
	E_PMLUnitMode.ePMLUnitMode_Production:
        CASE DescendantSequenceState OF
			0:
				NoStateTasksToComplete := FALSE;
				DescendantSequenceState := DescendantSequenceState + 10;
			10:
				StateTasksComplete := TRUE;
		END_CASE
		
	E_PMLUnitMode.ePMLUnitMode_Manual, E_PMLUnitMode.ePMLUnitMode_Maintenance:
        ;	
END_CASE

// Call Super
SUPER^.Unsuspending();
END_METHOD

END_FUNCTION_BLOCK

// ---- GlobalTextList.TcGTLO
TEXTLIST GlobalTextList
  685 = '%s'
  680 = 'Abort'
  11 = 'Aborted'
  86 = 'Aborting'
  452 = 'Clear'
  467 = 'Clearing'
  754 = 'Complete'
  302 = 'Completing'
  663 = 'Execute'
  51 = 'Held'
  744 = 'Hold'
  369 = 'Holding'
  342 = 'Idle'
  46 = 'Maintenance'
  904 = 'Manual'
  929 = 'Production'
  181 = 'Reset'
  123 = 'Resetting'
  639 = 'SC'
  77 = 'Start'
  888 = 'Starting'
  516 = 'State: %s'
  828 = 'Stop'
  796 = 'Stopped'
  161 = 'Stopping'
  806 = 'Suspend'
  623 = 'Suspended'
  229 = 'Suspending'
  782 = 'Un-Hold'
  466 = 'Un-Holding'
  901 = 'Un-Suspend'
  254 = 'Un-Suspending'
  197 = 'Unhold'
  832 = 'Unsuspend'
END_TEXTLIST
